{attribute wpf [Container(Layout.Stack)]}
FUNCTION_BLOCK TcoDoor EXTENDS TcoCore.TcoComponent IMPLEMENTS ITcoDoorLock
VAR_IN_OUT
    inoIsOpen : BOOL;
    inoIsLocked : BOOL;
    inoLock : BOOL;
END_VAR
VAR
    {attribute addProperty Name "<#Opened#>"}
    _isOpen : TcoElements.TcoDi(THIS^);

    {attribute addProperty Name "<#Locked#>"}
    _isLocked : TcoElements.TcoDi(THIS^);

    {attribute addProperty Name "<#Lock#>"}
    _lock : TcoElements.TcoDo(THIS^);


END_VAR

THIS^._isLocked(inoSignal :=  inoIsLocked);                    
THIS^._isOpen(inoSignal :=  inoIsOpen);                    
THIS^._lock(inoSignal   :=  inoLock);

PROPERTY IsClosed : BOOL
GET
IsClosed := THIS^._isOpen.IsFalse;
END_GET
END_PROPERTY

PROPERTY IsLocked : BOOL
GET
IsLocked := THIS^._isOpen.IsFalse and THIS^._isLocked.IsTrue ;
END_GET
END_PROPERTY

PROPERTY IsOpen : BOOL
GET
IsOpen := THIS^._isOpen.IsTrue;
END_GET
END_PROPERTY

METHOD Lock : BOOL
VAR_INPUT
END_VAR
Lock := FALSE;

THIS^._lock.Set();

IF	THIS^._isOpen.IsFalse THEN 
		
	IF THIS^._isLocked.IsTrue THEN 
		Lock := TRUE;
	END_IF
END_IF
END_METHOD

(*~
	<docu>
		<summary>
			Restores this instance to the Ready state. Can be called explicitly or from within one of the restore mechanisms.	
		</summary>			
	</docu>	
~*)
METHOD  Restore : ITcoRestorable
Unlock();
END_METHOD

(*~
	<docu>
		<summary>
		    Custom service (manual, maintenance) logic.
			This method must be implemented in derived class.
		</summary>			
	</docu>	
~*)
METHOD PROTECTED  ServiceMode
END_METHOD

METHOD UnLock : BOOL
VAR_INPUT
END_VAR

UnLock := FALSE;

THIS^._lock.Reset();
		
IF THIS^._isLocked.IsFalse THEN 
	UnLock := TRUE;
END_IF
END_METHOD

END_FUNCTION_BLOCK

(* stored: Version 1.1.0.1
   POU TcoDoor: Id {9ce8399f-b572-4d38-920f-7e58b0c9ce1c}, SpecialFunc None
   Property IsClosed: Id {92199df2-fdc3-4a20-b98f-2a2b6f3fc647}
   Get Get: Id {6e63724b-ab8e-456e-ba12-e37287c3c066}
   Property IsLocked: Id {2be8febe-191a-41ff-868b-ec3c2c82acb4}
   Get Get: Id {2524aa82-06c9-4835-80f9-105e58ef4c0e}
   Property IsOpen: Id {98b819b2-e2c3-40a5-ad00-0f54c1064163}
   Get Get: Id {8abeda15-a6e3-488c-8a7a-5b11b2469dd9}
   Method Lock: Id {2f6c419d-07f8-43d2-b213-d85628e6883c}
   Method Restore: Id {4f7bad87-7060-4350-8504-8df413b6f77b}
   Method ServiceMode: Id {27b1f781-c1bc-4474-b6db-2e6e98699307}
   Method UnLock: Id {8213b87e-87a1-408e-9a19-d9a09d05dac0} *)
